// TIA Portal project "Receptek" (V15.1)
// Harmadik projekt(13.-14. utolso laborok)

(* hardware
DEVICE "S7300/ET200M station_1"  S7-300 station
   slot 0: "Rail_0"  Rail  6ES7 390-1***0-0AA0
   slot 2: "PLC_1"  CPU 314C-2 PN/DP  6ES7 314-6EH04-0AB0  V3.3
      slot 2: "PROFINET interface_1"  PN-IO
         slot 1: "Port_1"  Port
         slot 2: "Port_2"  Port
      slot 5: "DI 24/DO 16_1"  DI24/DO16
      slot 6: "AI 5/AO 2_1"  AI5/AO2
      slot 7: "Count_1"  Counter
      slot 8: "Positioning_1"  Positioning
DEVICE "HMI_1"  KTP600 Basic color PN
   slot 0: "HMI_1"  KTP600 Basic color PN  6AV6 647-0AD11-3AX0  12.0.0.0
   slot 1: "HMI_RT_1"  KTP600 Basic color PN  6AV6 647-0AD11-3AX0  12.0.0.0
   slot 5: "HMI_1.IE_CP_1"  PROFINET Interface  12.0.0.0
      slot 1: "PROFINET Interface_1"  PROFINET Interface
         slot 1: "Port_1"  Port
*)

// ===== PLC "PLC_1"  CPU 314C-2 PN/DP =====

VAR_GLOBAL   // PLC tag table "Default tag table"
   "Recept_szam" AT %MW10 : Int;
   "address" AT %MD12 : DWord;
   "Kiolvasas_bit" AT %M20.0 : Bool;
   "Mentes_bit" AT %M20.1 : Bool;
   "Elozo_Recept_Szam" AT %MW12 : Int;
   "true" AT %M20.2 : Bool;
   "Elso_lefutas" AT %M20.3 : Bool;
END_VAR

DATA_BLOCK "Strukturak"   // DB1
{ S7_Optimized_Access := 'FALSE' }
VERSION : 0.1
   VAR
      RCP_ARRAY : Array[0..10] of Struct
         Nev : Word;
         Tej : Word;
         Viz : Word;
         Szinezo : Word;
         Cukor : Word;
      END_STRUCT;
      aktualis_nev : Word;
      aktualis_tej : Word;
      aktualis_viz : Word;
      aktualis_szinezo : Word;
      aktualis_cukor : Word;
   END_VAR
BEGIN
END_DATA_BLOCK

FUNCTION "load_RCP" : Void   // FC1, LAD
{ S7_Optimized_Access := 'FALSE' }
VERSION : 0.1
   VAR_TEMP
      address : DWord;
      offset : Word;
   END_VAR
BEGIN

REGION Network 1 (STL)
         L     "Recept_szam";
         L     10;
         *D;
         T     #offset;
         OPN   "Strukturak";
         L     P#0.0;
         L     #offset;
         SLD   3;
         +D;
         T     #address;
         L     DBW[#address];
         T     "Strukturak".aktualis_nev;
END_REGION

REGION Network 2 (STL)
         L     "Recept_szam";
         L     10;
         *D;
         L     2;
         +D;
         T     #offset;
         OPN   "Strukturak";
         L     P#0.0;
         L     #offset;
         SLD   3;
         +D;
         T     #address;
         L     DBW[#address];
         T     "Strukturak".aktualis_tej;
END_REGION

REGION Network 3 (STL)
         L     "Recept_szam";
         L     10;
         *D;
         L     4;
         +D;
         T     #offset;
         OPN   "Strukturak";
         L     P#0.0;
         L     #offset;
         SLD   3;
         +D;
         T     #address;
         L     DBW[#address];
         T     "Strukturak".aktualis_viz;
END_REGION

REGION Network 4 (STL)
         L     "Recept_szam";
         L     10;
         *D;
         L     6;
         +D;
         T     #offset;
         OPN   "Strukturak";
         L     P#0.0;
         L     #offset;
         SLD   3;
         +D;
         T     #address;
         L     DBW[#address];
         T     "Strukturak".aktualis_szinezo;
END_REGION

REGION Network 5 (STL)
         L     "Recept_szam";
         L     10;
         *D;
         L     8;
         +D;
         T     #offset;
         OPN   "Strukturak";
         L     P#0.0;
         L     #offset;
         SLD   3;
         +D;
         T     #address;
         L     DBW[#address];
         T     "Strukturak".aktualis_cukor;
END_REGION

REGION Network 6
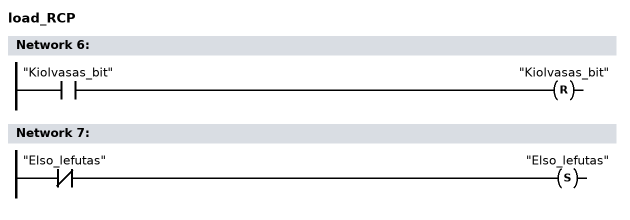
   RUNG wire#powerrail
      Contact( "Kiolvasas_bit" )
      R_Coil( "Kiolvasas_bit" )
   END_RUNG
   // the same network as SCL:
   IF "Kiolvasas_bit" THEN "Kiolvasas_bit" := FALSE; END_IF;
END_REGION

REGION Network 7
   RUNG wire#powerrail
      I_Contact( "Elso_lefutas" )
      S_Coil( "Elso_lefutas" )
   END_RUNG
   // the same network as SCL:
   IF NOT "Elso_lefutas" THEN "Elso_lefutas" := TRUE; END_IF;
END_REGION
END_FUNCTION

FUNCTION "Mentes" : Void   // FC2, LAD
{ S7_Optimized_Access := 'FALSE' }
VERSION : 0.1
   VAR_TEMP
      offset : Word;
      address : DWord;
   END_VAR
BEGIN

REGION Network 1 (STL)
   //menteshez
         L     "Recept_szam";
         L     10;
         *D;
         T     #offset;

         L     P#0.0;
         L     #offset;
         SLD   3;
         +D;
         OPN   "Strukturak";
         T     #address;
         L     "Strukturak".aktualis_nev;
         T     DBW [#address];
END_REGION

REGION Network 2 (STL)
         L     "Recept_szam";
         L     10;
         *D;
         L     2;
         +D;
         T     #offset;
         L     P#0.0;
         L     #offset;
         SLD   3;
         +D;
         OPN   "Strukturak";
         T     #address;
         L     "Strukturak".aktualis_tej;
         T     DBW [#address];
END_REGION

REGION Network 3 (STL)
         L     "Recept_szam";
         L     10;
         *D;
         L     4;
         +D;
         T     #offset;
         L     P#0.0;
         L     #offset;
         SLD   3;
         +D;
         OPN   "Strukturak";
         T     #address;
         L     "Strukturak".aktualis_viz;
         T     DBW [#address];
END_REGION

REGION Network 4 (STL)
         L     "Recept_szam";
         L     10;
         *D;
         L     6;
         +D;
         T     #offset;
         L     P#0.0;
         L     #offset;
         SLD   3;
         +D;
         OPN   "Strukturak";
         T     #address;
         L     "Strukturak".aktualis_szinezo;
         T     DBW [#address];
END_REGION

REGION Network 5 (STL)
         L     "Recept_szam";
         L     10;
         *D;
         L     8;
         +D;
         T     #offset;
         L     P#0.0;
         L     #offset;
         SLD   3;
         +D;
         OPN   "Strukturak";
         T     #address;
         L     "Strukturak".aktualis_cukor;
         T     DBW [#address];
END_REGION

REGION Network 6
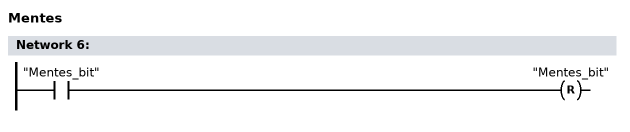
   RUNG wire#powerrail
      Contact( "Mentes_bit" )
      R_Coil( "Mentes_bit" )
   END_RUNG
   // the same network as SCL:
   IF "Mentes_bit" THEN "Mentes_bit" := FALSE; END_IF;
END_REGION
END_FUNCTION

ORGANIZATION_BLOCK "Main"   // OB1, LAD
TITLE = "Main Program Sweep (Cycle)"
{ S7_Optimized_Access := 'FALSE' }
VERSION : 0.1
   VAR_TEMP
      OB1_EV_CLASS : Byte;   // Bits 0-3 = 1 (Coming event), Bits 4-7 = 1 (Event class 1)
      OB1_SCAN_1 : Byte;   // 1 (Cold restart scan 1 of OB 1), 3 (Scan 2-n of OB 1)
      OB1_PRIORITY : Byte;   // Priority of OB Execution
      OB1_OB_NUMBR : Byte;   // 1 (Organization block 1, OB1)
      OB1_RESERVED_1 : Byte;   // Reserved for system
      OB1_RESERVED_2 : Byte;   // Reserved for system
      OB1_PREV_CYCLE : Int;   // Cycle time of previous OB1 scan (milliseconds)
      OB1_MIN_CYCLE : Int;   // Minimum cycle time of OB1 (milliseconds)
      OB1_MAX_CYCLE : Int;   // Maximum cycle time of OB1 (milliseconds)
      OB1_DATE_TIME : Date_And_Time;   // Date and time OB1 started
   END_VAR
BEGIN

REGION Network 1
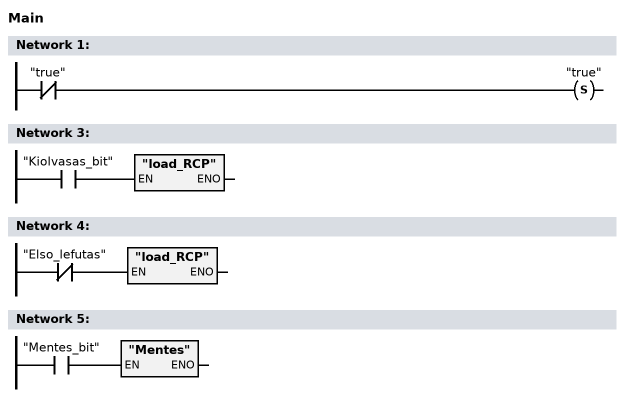
   RUNG wire#powerrail
      I_Contact( "true" )
      S_Coil( "true" )
   END_RUNG
   // the same network as SCL:
   IF NOT "true" THEN "true" := TRUE; END_IF;
END_REGION

REGION Network 2 (STL)
         L     "Recept_szam";
         L     "Elozo_Recept_Szam";
         <>I;
         JC    beiras;
         JU    vege;

   beiras:A     "true";
         =     "Kiolvasas_bit";
         L     "Recept_szam";
         L     10;
         <I;
         JC    ellenorzes;
         JU    tiz;

   ellenorzes:L     "Recept_szam";
         L     0;
         >I;
         JC    betoltes;
         JU    nulla;
   betoltes:L     "Recept_szam";
         T     "Elozo_Recept_Szam";
         JU    vege;


   nulla:L     0;
         T     "Recept_szam";
         T     "Elozo_Recept_Szam";
         JU    vege;
   tiz:  L     10;
         T     "Recept_szam";
         T     "Elozo_Recept_Szam";
         JU    vege;

   vege: NOP   0;
END_REGION

REGION Network 3
   RUNG wire#powerrail
      Contact( "Kiolvasas_bit" )
      "load_RCP"()
   END_RUNG
   // the same network as SCL:
   IF "Kiolvasas_bit" THEN "load_RCP"(); END_IF;
END_REGION

REGION Network 4
   RUNG wire#powerrail
      I_Contact( "Elso_lefutas" )
      "load_RCP"()
   END_RUNG
   // the same network as SCL:
   IF NOT "Elso_lefutas" THEN "load_RCP"(); END_IF;
END_REGION

REGION Network 5
   RUNG wire#powerrail
      Contact( "Mentes_bit" )
      "Mentes"()
   END_RUNG
   // the same network as SCL:
   IF "Mentes_bit" THEN "Mentes"(); END_IF;
END_REGION
END_ORGANIZATION_BLOCK

(* ===== HMI "HMI_RT_1" =====
system functions are stored by id; their names below are inferred from use
connection "HMI_Connection_1": ETHERNET, SIMATIC S7 300/400 MPI

HMI tags "Default tag table"
   "Tag_ScreenNumber" : UInt, internal
   "Recept_szam" : Int = PLC Recept_szam AT %MW10, 1 s
   "Strukturak_aktualis_nev" : Word = PLC Strukturak.aktualis_nev AT %DB1.DBW110, 1 s
   "Strukturak_aktualis_tej" : Word = PLC Strukturak.aktualis_tej AT %DB1.DBW112, 1 s
   "Strukturak_aktualis_viz" : Word = PLC Strukturak.aktualis_viz AT %DB1.DBW114, 1 s
   "Strukturak_aktualis_szinezo" : Word = PLC Strukturak.aktualis_szinezo AT %DB1.DBW116, 1 s
   "Strukturak_aktualis_cukor" : Word = PLC Strukturak.aktualis_cukor AT %DB1.DBW118, 1 s
   "Kiolvasas_bit" : Bool = PLC Kiolvasas_bit AT %M20.0, 1 s
   "Mentes_bit" : Bool = PLC Mentes_bit AT %M20.1, 1 s

Template "Template_1" 320x240
   Button "Exit" at 266,202 size 52x37; TextOff 'Exit'; PictureOff "ExitRuntime_KTP600_Basic_color_PN"; PictureOn "ExitRuntime_KTP600_Basic_color_PN"
      on Release: StopRuntime(0)
   Button "Template_Button" at 213,202 size 52x37; TextOff 'Text'
   Button "Template_Button_1" at 160,202 size 52x37; TextOff 'Text'
   Button "Template_Button_2" at 107,202 size 52x37; TextOff 'Indi.Cim.'
      on Press: ActivateScreen("Indirekt_cimzes", 0)
   Button "Alarms" at 54,202 size 52x37; TextOff 'Alarms'; PictureOff "AlarmDisplay_KTP600_Basic_color_PN"; PictureOn "AlarmDisplay_KTP600_Basic_color_PN"
      on Release: function_ef3f5d25("Alarm window_Unacknowledged", -1)
   Button "Start screen" at 1,202 size 52x37; TextOff 'Start screen'; PictureOff "NavigateHome_KTP600_Basic_color_PN"; PictureOn "NavigateHome_KTP600_Basic_color_PN"
      on Release: ActivateScreen("Root screen", 0)
   SymbolicIOField "Symbolic_IO_Field_Screen" at 69,7 size 164x24; TextOff '0'; TextOn '1'; TextList "TextList_ScreenNames"
      ProcessValue <- "Tag_ScreenNumber"
      on Change: ActivateScreenByNumber("Tag_ScreenNumber", 0)
   DateTimeField "HmiScreenItemData" at 235,19 size 85x19
   DateTimeField "HmiScreenItemData_1" at 235,0 size 85x19
   GraphicView "Logo" at 0,0 size 67x38; Picture "Logo of HMI_1"

screen "Root screen" 320x240, template "Template_1"
   on GenerateScreen: SetTag("Tag_ScreenNumber", 1)
   TextField "HmiScreenItemData" at 32,109 size 256x17; Text 'Welcome to HMI_1 (KTP600 Basic color PN)!'

screen "Indirekt_cimzes" 320x240
   IOField "I/O field_1" at 10,36 size 96x23; FormatPattern s99
      ProcessValue <- "Recept_szam"
   TextField "Text field_1" at 116,36 size 203x13; Text 'Hanyadik receptet kivanjuk modositani?'
   IOField "I/O field_2" at 11,60 size 96x23; FormatPattern 99999
      ProcessValue <- "Strukturak_aktualis_nev"
   IOField "I/O field_3" at 12,83 size 96x23; FormatPattern 99999
      ProcessValue <- "Strukturak_aktualis_tej"
   IOField "I/O field_4" at 12,107 size 96x23; FormatPattern 99999
      ProcessValue <- "Strukturak_aktualis_viz"
   IOField "I/O field_5" at 13,129 size 96x23; FormatPattern 99999
      ProcessValue <- "Strukturak_aktualis_szinezo"
   IOField "I/O field_6" at 11,155 size 96x23; FormatPattern 99999
      ProcessValue <- "Strukturak_aktualis_cukor"
   TextField "Text field_2" at 116,61 size 22x15; Text 'NEV'
   TextField "Text field_3" at 118,84 size 21x15; Text 'TEJ'
   TextField "Text field_4" at 122,112 size 21x15; Text 'VIZ'
   TextField "Text field_5" at 116,140 size 49x15; Text 'SZINEZO'
   TextField "Text field_6" at 112,163 size 40x15; Text 'CUKOR'
   TextField "Text field_7" at 12,8 size 140x20; Text 'INDIREKT CIMZES'
   Button "Button_1" at 176,55 size 124x43; TextOff 'Értékek vissza állítása'
      on Press: SetBit("Kiolvasas_bit")
   Button "Button_2" at 176,112 size 124x40; TextOff 'Mentés'
      on Press: SetBit("Mentes_bit")
   Button "Exit" at 266,202 size 52x37; TextOn 'Exit'; TextOff 'Exit'; PictureOn "ExitRuntime_KTP600_Basic_color_PN"; PictureOff "ExitRuntime_KTP600_Basic_color_PN"
      on Release: StopRuntime(0)
   Button "Template_Button" at 213,202 size 52x37; TextOff 'Text'
   Button "Template_Button_1" at 160,202 size 52x37; TextOff 'Text'
   Button "Template_Button_2" at 107,202 size 52x37; TextOff 'Indi.Cim.'
      on Press: ActivateScreen("Indirekt_cimzes", 0)
   Button "Alarms" at 54,202 size 52x37; TextOn 'Alarms'; TextOff 'Alarms'; PictureOn "AlarmDisplay_KTP600_Basic_color_PN"; PictureOff "AlarmDisplay_KTP600_Basic_color_PN"
      on Release: function_ef3f5d25("Alarm window_Unacknowledged", -1)
   Button "Start screen" at 1,202 size 52x37; TextOn 'Start screen'; TextOff 'Start screen'; PictureOn "NavigateHome_KTP600_Basic_color_PN"; PictureOff "NavigateHome_KTP600_Basic_color_PN"
      on Release: ActivateScreen("Root screen", 0)
*)